FUNCTION_BLOCK PnpCylindersBA (* Composite Function Block Type *)
  (* Standard: 61499-2 *)
  (* Version 0.2, 2003-12-05, JHC, Rockwell Automation, Renamed from NEWCOMPFB. *)
  (* Version 0.1, 2002-01-08, JHC, Rockwell Automation, Added DLY FB as example. *)
  (* Version 0.0, 2000-05-27, JHC, Rockwell Automation *)
  (* Compiler header: package fb.rt.pnp; *)
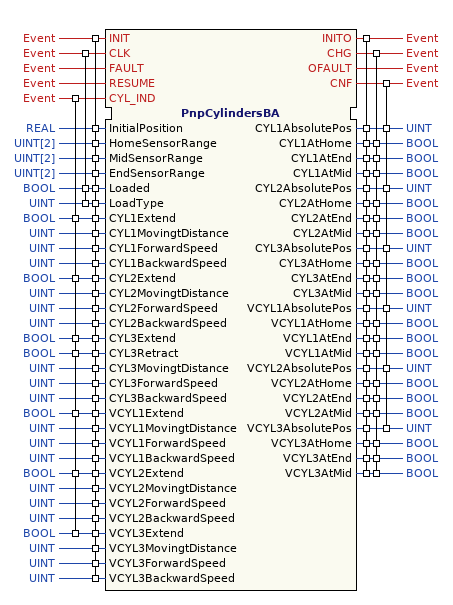
  EVENT_INPUT
    INIT WITH HomeSensorRange, EndSensorRange, InitialPosition, LoadType, Loaded, MidSensorRange, CYL1Extend, CYL2Extend, CYL3Extend, CYL3Retract, VCYL1Extend, VCYL2Extend, VCYL3Extend, CYL1MovingtDistance, CYL1ForwardSpeed, CYL1BackwardSpeed, CYL2MovingtDistance, CYL2ForwardSpeed, CYL2BackwardSpeed, CYL3MovingtDistance, CYL3ForwardSpeed, CYL3BackwardSpeed, VCYL1MovingtDistance, VCYL1ForwardSpeed, VCYL1BackwardSpeed, VCYL2MovingtDistance, VCYL2ForwardSpeed, VCYL3MovingtDistance, VCYL3ForwardSpeed, VCYL3BackwardSpeed, VCYL2BackwardSpeed; (* Initialization Request *)
    CLK WITH LoadType, Loaded;
    FAULT;
    RESUME;
    CYL_IND WITH CYL1Extend, CYL2Extend, CYL3Extend, CYL3Retract, VCYL1Extend, VCYL2Extend, VCYL3Extend;
  END_EVENT
  EVENT_OUTPUT
    INITO WITH CYL1AbsolutePos, CYL1AtHome, CYL1AtEnd, CYL1AtMid, CYL2AbsolutePos, CYL2AtHome, CYL2AtEnd, CYL2AtMid, CYL3AbsolutePos, CYL3AtHome, CYL3AtEnd, CYL3AtMid, VCYL1AbsolutePos, VCYL1AtHome, VCYL1AtEnd, VCYL1AtMid, VCYL2AbsolutePos, VCYL2AtHome, VCYL2AtEnd, VCYL2AtMid, VCYL3AbsolutePos, VCYL3AtHome, VCYL3AtEnd, VCYL3AtMid; (* Initialization Confirm *)
    CHG WITH CYL1AtHome, CYL1AtEnd, CYL1AtMid, CYL2AtHome, CYL2AtEnd, CYL2AtMid, CYL3AtHome, CYL3AtEnd, CYL3AtMid, VCYL1AtHome, VCYL1AtEnd, VCYL1AtMid, VCYL2AtHome, VCYL2AtEnd, VCYL2AtMid, VCYL3AtHome, VCYL3AtEnd, VCYL3AtMid;
    OFAULT;
    CNF WITH CYL1AbsolutePos, CYL2AbsolutePos, CYL3AbsolutePos, VCYL1AbsolutePos, VCYL2AbsolutePos, VCYL3AbsolutePos;
  END_EVENT
  VAR_INPUT
    InitialPosition : REAL; (* Initial position *)
    HomeSensorRange : ARRAY [0..1] OF UINT; (* Detection range of home sensor *)
    MidSensorRange : ARRAY [0..1] OF UINT; (* Detection range of home sensor *)
    EndSensorRange : ARRAY [0..1] OF UINT; (* Detection range of end sensor *)
    Loaded : BOOL;
    LoadType : UINT;
    CYL1Extend : BOOL;
    CYL1MovingtDistance : UINT;
    CYL1ForwardSpeed : UINT;
    CYL1BackwardSpeed : UINT;
    CYL2Extend : BOOL;
    CYL2MovingtDistance : UINT;
    CYL2ForwardSpeed : UINT;
    CYL2BackwardSpeed : UINT;
    CYL3Extend : BOOL;
    CYL3Retract : BOOL;
    CYL3MovingtDistance : UINT;
    CYL3ForwardSpeed : UINT;
    CYL3BackwardSpeed : UINT;
    VCYL1Extend : BOOL;
    VCYL1MovingtDistance : UINT;
    VCYL1ForwardSpeed : UINT;
    VCYL1BackwardSpeed : UINT;
    VCYL2Extend : BOOL;
    VCYL2MovingtDistance : UINT;
    VCYL2ForwardSpeed : UINT;
    VCYL2BackwardSpeed : UINT;
    VCYL3Extend : BOOL;
    VCYL3MovingtDistance : UINT;
    VCYL3ForwardSpeed : UINT;
    VCYL3BackwardSpeed : UINT;
  END_VAR
  VAR_OUTPUT
    CYL1AbsolutePos : UINT; (* Current position *)
    CYL1AtHome : BOOL; (* Detected at home position *)
    CYL1AtEnd : BOOL; (* Detected at end position *)
    CYL1AtMid : BOOL;
    CYL2AbsolutePos : UINT; (* Current position *)
    CYL2AtHome : BOOL; (* Detected at home position *)
    CYL2AtEnd : BOOL; (* Detected at end position *)
    CYL2AtMid : BOOL;
    CYL3AbsolutePos : UINT; (* Current position *)
    CYL3AtHome : BOOL; (* Detected at home position *)
    CYL3AtEnd : BOOL; (* Detected at end position *)
    CYL3AtMid : BOOL;
    VCYL1AbsolutePos : UINT; (* Current position *)
    VCYL1AtHome : BOOL; (* Detected at home position *)
    VCYL1AtEnd : BOOL; (* Detected at end position *)
    VCYL1AtMid : BOOL;
    VCYL2AbsolutePos : UINT; (* Current position *)
    VCYL2AtHome : BOOL; (* Detected at home position *)
    VCYL2AtEnd : BOOL; (* Detected at end position *)
    VCYL2AtMid : BOOL;
    VCYL3AbsolutePos : UINT; (* Current position *)
    VCYL3AtHome : BOOL; (* Detected at home position *)
    VCYL3AtEnd : BOOL; (* Detected at end position *)
    VCYL3AtMid : BOOL;
  END_VAR
  FBS
    CYL1 : GenericCylinderModelType2;
    CYL2 : GenericCylinderModelType2;
    CYL3 : GenericCylinderModelType1;
    VCYL1 : GenericCylinderModelType2;
    VCYL2 : GenericCylinderModelType2;
    VCYL3 : GenericCylinderModelType2;
  END_FBS
  EVENT_CONNECTIONS
    INIT TO CYL1.INIT;
    CYL1.INITO TO CYL2.INIT;
    CYL2.INITO TO CYL3.INIT;
    CYL3.INITO TO VCYL1.INIT;
    VCYL1.INITO TO VCYL2.INIT;
    VCYL2.INITO TO VCYL3.INIT;
    VCYL3.INITO TO INITO;
    VCYL3.OFAULT TO OFAULT;
    VCYL2.OFAULT TO VCYL3.FAULT;
    VCYL1.OFAULT TO VCYL2.FAULT;
    CYL2.OFAULT TO CYL3.FAULT;
    CYL1.OFAULT TO CYL2.FAULT;
    FAULT TO CYL1.FAULT;
    CLK TO CYL1.CLK;
    CLK TO CYL2.CLK;
    CLK TO CYL3.CLK;
    CLK TO VCYL1.CLK;
    CLK TO VCYL2.CLK;
    CLK TO VCYL3.CLK;
    CYL1.CHG TO CHG;
    CYL2.CHG TO CHG;
    CYL3.CHG TO CHG;
    VCYL1.CHG TO CHG;
    VCYL2.CHG TO CHG;
    VCYL3.CHG TO CHG;
    VCYL3.CNF TO CNF;
    VCYL2.CNF TO CNF;
    VCYL1.CNF TO CNF;
    CYL3.CNF TO CNF;
    CYL2.CNF TO CNF;
    CYL1.CNF TO CNF;
    RESUME TO CYL1.RESUME;
    RESUME TO CYL2.RESUME;
    RESUME TO CYL3.RESUME;
    RESUME TO VCYL1.RESUME;
    RESUME TO VCYL2.RESUME;
    RESUME TO VCYL3.RESUME;
    CYL_IND TO VCYL3.CYL_IND;
    CYL_IND TO CYL1.CYL_IND;
    CYL_IND TO CYL2.CYL_IND;
    CYL_IND TO CYL3.CYL_IND;
    CYL_IND TO VCYL1.CYL_IND;
    CYL_IND TO VCYL2.CYL_IND;
    CYL3.OFAULT TO VCYL1.FAULT;
  END_CONNECTIONS
  DATA_CONNECTIONS
    HomeSensorRange TO CYL1.HomeSensorRange;
    HomeSensorRange TO CYL2.HomeSensorRange;
    HomeSensorRange TO CYL3.HomeSensorRange;
    HomeSensorRange TO VCYL1.HomeSensorRange;
    HomeSensorRange TO VCYL2.HomeSensorRange;
    HomeSensorRange TO VCYL3.HomeSensorRange;
    MidSensorRange TO VCYL3.MidSensorRange;
    MidSensorRange TO CYL1.MidSensorRange;
    MidSensorRange TO CYL2.MidSensorRange;
    MidSensorRange TO CYL3.MidSensorRange;
    MidSensorRange TO VCYL1.MidSensorRange;
    MidSensorRange TO VCYL2.MidSensorRange;
    EndSensorRange TO CYL1.EndSensorRange;
    EndSensorRange TO CYL2.EndSensorRange;
    EndSensorRange TO CYL3.EndSensorRange;
    EndSensorRange TO VCYL1.EndSensorRange;
    EndSensorRange TO VCYL2.EndSensorRange;
    EndSensorRange TO VCYL3.EndSensorRange;
    InitialPosition TO CYL1.InitialPosition;
    InitialPosition TO CYL2.InitialPosition;
    InitialPosition TO CYL3.InitialPosition;
    InitialPosition TO VCYL1.InitialPosition;
    InitialPosition TO VCYL2.InitialPosition;
    InitialPosition TO VCYL3.InitialPosition;
    Loaded TO CYL1.Loaded;
    Loaded TO CYL2.Loaded;
    Loaded TO CYL3.Loaded;
    Loaded TO VCYL1.Loaded;
    Loaded TO VCYL2.Loaded;
    Loaded TO VCYL3.Loaded;
    LoadType TO CYL1.LoadType;
    LoadType TO CYL2.LoadType;
    LoadType TO CYL3.LoadType;
    LoadType TO VCYL1.LoadType;
    LoadType TO VCYL2.LoadType;
    LoadType TO VCYL3.LoadType;
    CYL1Extend TO CYL1.Extend;
    CYL2Extend TO CYL2.Extend;
    CYL3Extend TO CYL3.Extend;
    CYL3Retract TO CYL3.Retract;
    VCYL1Extend TO VCYL1.Extend;
    VCYL2Extend TO VCYL2.Extend;
    VCYL3Extend TO VCYL3.Extend;
    VCYL1ForwardSpeed TO VCYL1.ForwardSpeed;
    VCYL1BackwardSpeed TO VCYL1.BackwardSpeed;
    VCYL1MovingtDistance TO VCYL1.MovingtDistance;
    VCYL2ForwardSpeed TO VCYL2.ForwardSpeed;
    VCYL2BackwardSpeed TO VCYL2.BackwardSpeed;
    VCYL2MovingtDistance TO VCYL2.MovingtDistance;
    VCYL2MovingtDistance TO VCYL3.MovingtDistance;
    VCYL1BackwardSpeed TO VCYL3.BackwardSpeed;
    VCYL1ForwardSpeed TO VCYL3.ForwardSpeed;
    CYL3MovingtDistance TO CYL3.MovingtDistance;
    CYL3BackwardSpeed TO CYL3.BackwardSpeed;
    CYL3ForwardSpeed TO CYL3.ForwardSpeed;
    CYL2ForwardSpeed TO CYL2.ForwardSpeed;
    CYL2BackwardSpeed TO CYL2.BackwardSpeed;
    CYL2MovingtDistance TO CYL2.MovingtDistance;
    CYL1MovingtDistance TO CYL1.MovingtDistance;
    CYL1BackwardSpeed TO CYL1.BackwardSpeed;
    CYL1ForwardSpeed TO CYL1.ForwardSpeed;
    CYL1.AbsolutePos TO CYL1AbsolutePos;
    CYL2.AbsolutePos TO CYL2AbsolutePos;
    CYL3.AbsolutePos TO CYL3AbsolutePos;
    VCYL1.AbsolutePos TO VCYL1AbsolutePos;
    VCYL2.AbsolutePos TO VCYL2AbsolutePos;
    VCYL3.AbsolutePos TO VCYL3AbsolutePos;
    CYL1.AtHome TO CYL1AtHome;
    CYL1.AtEnd TO CYL1AtEnd;
    CYL1.AtMid TO CYL1AtMid;
    CYL2.AtHome TO CYL2AtHome;
    CYL2.AtEnd TO CYL2AtEnd;
    CYL2.AtMid TO CYL2AtMid;
    CYL3.AtHome TO CYL3AtHome;
    CYL3.AtEnd TO CYL3AtEnd;
    CYL3.AtMid TO CYL3AtMid;
    VCYL1.AtHome TO VCYL1AtHome;
    VCYL1.AtEnd TO VCYL1AtEnd;
    VCYL1.AtMid TO VCYL1AtMid;
    VCYL2.AtHome TO VCYL2AtHome;
    VCYL2.AtEnd TO VCYL2AtEnd;
    VCYL2.AtMid TO VCYL2AtMid;
    VCYL3.AtHome TO VCYL3AtHome;
    VCYL3.AtEnd TO VCYL3AtEnd;
    VCYL3.AtMid TO VCYL3AtMid;
  END_CONNECTIONS
END_FUNCTION_BLOCK
